TEXTLIST TextList_1_20_Speed
  1 = '1'
  2 = '2'
  3 = '3'
  4 = '4'
  5 = '5'
  6 = '6'
  7 = '7'
  8 = '8'
  9 = '9'
  10 = '10'
  11 = '11'
  12 = '12'
  13 = '13'
  14 = '14'
  15 = '15'
  16 = '16'
  17 = '17'
  18 = '18'
  19 = '19'
  20 = '20'
   = ''
END_TEXTLIST

(* stored: Version 1.1.0.1, ProductVersion 3.1.4024.12
   TextList TextList_1_20_Speed: Id {05f66ab1-cdef-4e98-b34b-4536d8da2998} *)
